# EPICS autosave request: iocs/pncsIOC/iocBoot/iocPNCS/auto_settings.req
file "ADPNDetectorCXC_settings.req",  P=$(P),  R=cam1:
file "NDStdArrays_settings.req",  P=$(P),  R=image1:
file "commonPlugin_settings.req", P=$(P)
